% RSLogix 500 project oil flow.RSS, saved by version 8.30.00.16 %
PROJECT "UNTITLED"    % processor: Bul.1763 MicroLogix 1100 Series B %

PROGRAM FILES
  LAD 2 "MAIN"  6 rungs

DATA FILES
  O0 OUTPUT  4 elements
  I1 INPUT  6 elements
  S2 STATUS  66 elements
  B3 BINARY  1 elements
  T4 TIMER  2 elements
  C5 COUNTER  1 elements
  R6 CONTROL  1 elements
  N7 INTEGER  2 elements
  F8 FLOAT  2 elements

LADDER 2 "MAIN"
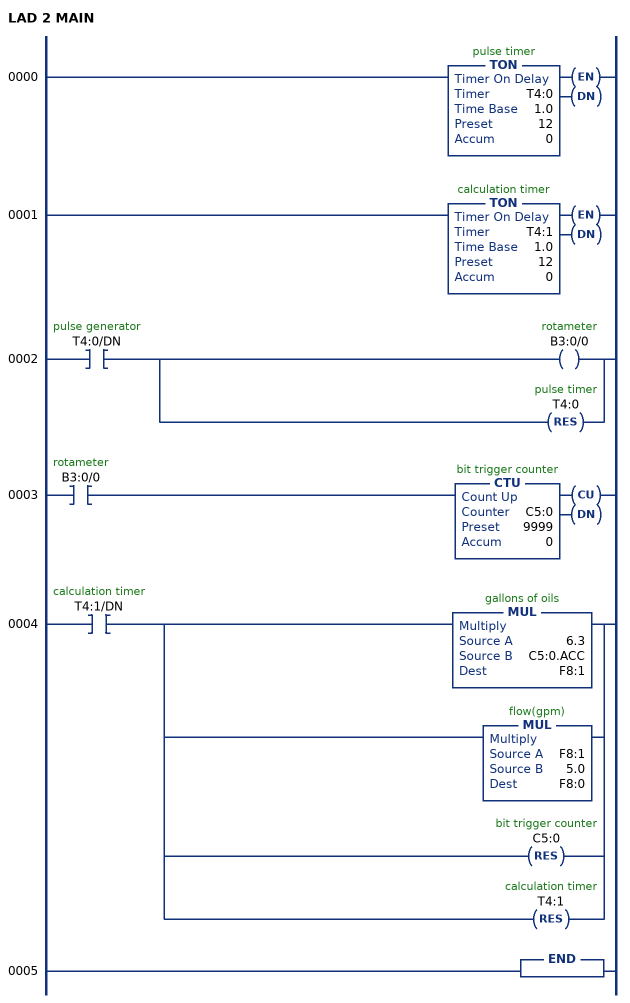
% Rung: 0 %
SOR TON T4:0 1.0 12 0 EOR
%   T4:0  "pulse timer" %
% Rung: 1 %
SOR TON T4:1 1.0 12 0 EOR
%   T4:1  "calculation timer" %
% Rung: 2 %
SOR XIC T4:0/DN BST OTE B3:0/0 NXB RES T4:0 BND EOR
%   T4:0/DN  "pulse generator" %
%   B3:0/0  "rotameter" %
%   T4:0  "pulse timer" %
% Rung: 3 %
SOR XIC B3:0/0 CTU C5:0 9999 0 EOR
%   B3:0/0  "rotameter" %
%   C5:0  "bit trigger counter" %
% Rung: 4 %
SOR XIC T4:1/DN BST MUL 6.3 C5:0.ACC F8:1 NXB MUL F8:1 5.0 F8:0 NXB RES C5:0 NXB RES T4:1 BND EOR
%   T4:1  "calculation timer" %
%   C5:0  "bit trigger counter" %
%   F8:1  "gallons of oils" %
%   F8:0  "flow(gpm)" %
% Rung: 5 %
SOR END EOR

OTHER DOCUMENTED ADDRESSES
  B3:0/1  "ons"
  I:0.0/0  "power on"
  N7:0  "total bit"
  N7:0/0  "total bit"
  N7:0/1  "adding bit"
  N7:1  "adding bit"

DATA TABLE (non-zero values as saved)
DATA T4
% .PRE .ACC %
% T4:0 % 12 0
% T4:1 % 12 0
DATA C5
% .PRE .ACC %
% C5:0 % 9999 0
DATA N7
% N7:0 % 197 1
